FUNCTION_BLOCK FB_AlarmEventSet
VAR_INPUT
	bAlarmEventTrigger:BOOL;
	tSetDelay:TIME;
	tResetDelay:TIME;
	bManualReset:BOOL;
	bResetError:BOOL;
	bEnableAlarm:BOOL;
END_VAR
VAR_OUTPUT
	bOutAlarmEvent:	BOOL;
END_VAR
VAR
	
	bReset:BOOL;
	TON_SetDelay:TON;
	TON_ResetDelay:TOF;
	Latch:SR;
END_VAR

IF (bManualReset AND bResetError AND NOT(bAlarmEventTrigger))
	OR (NOT(bManualReset) AND NOT(bAlarmEventTrigger))  OR NOT(bEnableAlarm) THEN
	bReset:=1;
ELSE
	bReset:=0;
END_IF

Latch(SET1:=TON_SetDelay.Q , 
	  RESET:=bReset , 
	  Q1=> );

TON_ResetDelay(IN:=Latch.Q1 , PT:=tResetDelay , Q=> , ET=> );
TON_SetDelay(IN:=bAlarmEventTrigger AND bEnableAlarm, PT:=tSetDelay , Q=> , ET=> );

bOutAlarmEvent:=TON_ResetDelay.Q;

END_FUNCTION_BLOCK

(* stored: Version 1.1.0.1, ProductVersion 3.1.4024.11
   POU FB_AlarmEventSet: Id {9a118d40-c5aa-4df4-aa51-269f418c9e9d}, SpecialFunc None *)
